// TIA Portal V20 export
DATA_BLOCK "Config"   // DB162
// stored: MemoryReserve 100, Namespace Unit1.Em1
   VAR
      em : "LAF_typeEmConfiguration";   // Configuration of EM Parameters
      cmStacker2NgBoxDetect : "LBC_typeDigitalSignalConfiguration";
      cmStacker2NgBoxFullDetect : "LBC_typeDigitalSignalConfiguration";
      cmStacker2NgBoxLoadingUpDown : "LBC_typeTwoWayActuatorConfiguration";
      cmStacker2NgBoxUnitMoverBwdFwd : "LBC_typeTwoWayActuatorConfiguration";
      cmStacker2NgBoxClampLeftOpenClose : "LBC_typeTwoWayActuatorConfiguration";
      cmStacker2NgBoxClampRightOpenClose : "LBC_typeTwoWayActuatorConfiguration";
      cmStacker2NgBoxClampMoverOpenClose : "LBC_typeTwoWayActuatorConfiguration";
      cmStacker2NgBoxLiftDownUp : "LBC_typeTwoWayActuatorConfiguration";
      cmStacker2NgBoxLockDownUp : "LBC_typeTwoWayActuatorConfiguration";
   END_VAR
BEGIN
   em.referenceDesignator.parent := WSTRING#'U1';
   em.referenceDesignator.relative := WSTRING#'EM0';
   cmStacker2NgBoxLoadingUpDown.referenceDesignator := WSTRING#'STACK NG CLAMP Z-AXIS';
   cmStacker2NgBoxLoadingUpDown.monitoringDiscrepancy := T#5s;
   cmStacker2NgBoxUnitMoverBwdFwd.referenceDesignator := WSTRING#'NG CLAMP UNIT MOVER';
   cmStacker2NgBoxUnitMoverBwdFwd.monitoringLeavingFeedback := T#10s;
   cmStacker2NgBoxUnitMoverBwdFwd.monitoringReachingFeedback := T#10s;
   cmStacker2NgBoxUnitMoverBwdFwd.monitoringDiscrepancy := T#5s;
   cmStacker2NgBoxClampLeftOpenClose.referenceDesignator := WSTRING#'STACK NG CLAMP LEFT';
   cmStacker2NgBoxClampLeftOpenClose.monitoringDiscrepancy := T#5s;
   cmStacker2NgBoxClampRightOpenClose.referenceDesignator := WSTRING#'STACK NG CLAMP RIGHT';
   cmStacker2NgBoxClampRightOpenClose.monitoringDiscrepancy := T#5s;
   cmStacker2NgBoxClampMoverOpenClose.referenceDesignator := WSTRING#'STACK NG CLAMP MOVER';
   cmStacker2NgBoxClampMoverOpenClose.monitoringDiscrepancy := T#5s;
   cmStacker2NgBoxLiftDownUp.referenceDesignator := WSTRING#'STACK NG BOX LIFT';
   cmStacker2NgBoxLiftDownUp.monitoringDiscrepancy := T#5s;
   cmStacker2NgBoxLockDownUp.referenceDesignator := WSTRING#'STACK NG BOX LOCK';
   cmStacker2NgBoxLockDownUp.monitoringDiscrepancy := T#5s;
END_DATA_BLOCK
